// TIA Portal V20 export
TYPE "typeSequenceControlNodeJobInterface"
// stored: Namespace Unit1.Em0
   STRUCT
      loadJob2 : "LER_typeJobInterface";
      unloadJob3 : "LER_typeJobInterface";
   END_STRUCT;
END_TYPE
